INTERFACE IGHT

{attribute 'object_name' := 'Clear'}
METHOD Clear : BOOL
VAR_INPUT
	bolFreePointer: BOOL;
END_VAR
END_METHOD

{attribute 'object_name' := 'Initialize'}
METHOD Initialize : BOOL
END_METHOD

PROPERTY Count : UINT
GET
END_GET
END_PROPERTY

{attribute 'object_name' := 'Lookup'}
METHOD Lookup : POINTER TO BYTE
VAR_INPUT
	uliKey: ULINT;
	bolRemove: BOOL;
END_VAR
END_METHOD

{attribute 'object_name' := 'AddItem'}
METHOD AddItem : BOOL
VAR_INPUT
	uliKey: ULINT;
	pData: POINTER TO BYTE;
END_VAR
END_METHOD

END_INTERFACE

(* stored: Version 1.1.0.1, ProductVersion 3.1.0.36
   Itf IGHT: Id {1369cddd-21ca-4288-aafc-6b12aed90293}
   Method Clear: Id {2b5f83c9-7e25-4125-ad11-d67fee5836df}
   Method Initialize: Id {43adaa89-a44f-4bbe-9e5c-4fae0639e37e}
   Property Count: Id {5bac76e5-ef0e-4aee-b32a-c5fdd14d0d2c}
   Get Get: Id {6b0d386d-80ac-4d44-89ca-d43d1bb95ffe}
   Method Lookup: Id {8fb41088-b237-4034-bdc0-99530f1c464b}
   Method AddItem: Id {9fe970a3-1a2e-4d3f-b649-fa00d84995e2} *)
